# B&R Automation Studio project Morozov_Lab
Automation Studio 

## Logical view

### Library Logical/Libraries/Library (ANSIC)

#### Library.fun - Exported functions and function blocks
```iecst
FUNCTION_BLOCK FB_Controller (*Функциональный блок регулятора*)
	VAR_INPUT
		e : REAL; (*Вход регулятора (об/мин)*)
	END_VAR
	VAR_OUTPUT
		u : REAL; (*Выход регулятора (В)*)
	END_VAR
	VAR
		dt : REAL; (*Шаг интегрирвоания (с)*)
		k_i : REAL; (*Интегральный коэфффициент*)
		k_p : REAL; (*Пропорциональный коэффициент*)
		max_abs_value : REAL; (*Максимальное входное напряжение*)
		integrator : FB_Integrator; (*ФБ-интератор в составе регулятора*)
		iyOld : REAL; (*Разница между выходом регулятора*)
	END_VAR
END_FUNCTION_BLOCK

FUNCTION_BLOCK FB_Integrator (*Функциональный блок интегратора*)
	VAR_INPUT
		in : REAL; (*Вход интеграторируещего звена*)
	END_VAR
	VAR_OUTPUT
		out : REAL; (*Выход интеграторируещего звена*)
	END_VAR
	VAR
		dt : REAL; (*Шаг интегрирования*)
		state : REAL; (*Состояние интегратора на*)
	END_VAR
END_FUNCTION_BLOCK

FUNCTION_BLOCK FB_Motor (*Функциональный блок двигателя*)
	VAR_INPUT
		in : REAL; (*Входное напряжение (В)*)
	END_VAR
	VAR_OUTPUT
		out_w : REAL; (*Частота вращения (об/мин)*)
	END_VAR
	VAR
		dt : REAL; (*Шаг интегрирования (с)*)
		k_e : REAL; (*Постоянная ЭДС двигателя*)
		T_m : REAL; (*Электромеханическая постоянная двигателя*)
		integrator : FB_Integrator; (*ФБ-интегратор в составе двигателя*)
	END_VAR
END_FUNCTION_BLOCK
```

#### FB_Motor.c
```c
#include <bur/plctypes.h>
#ifdef __cplusplus
	extern "C"
	{
#endif
	#include "Library.h"
#ifdef __cplusplus
	};
#endif
/* function block for motors model */
void FB_Motor(struct FB_Motor* inst)
{
	REAL a = inst->in / inst->k_e - inst->out_w;
	REAL b = a / inst->T_m;

	inst->integrator.in = b;
	FB_Integrator(&inst->integrator);

	inst->out_w = inst->integrator.out;
}
```

#### FB_Integrator.c
```c
#include <bur/plctypes.h>
#ifdef __cplusplus
	extern "C"
	{
#endif
	#include "Library.h"
#ifdef __cplusplus
	};
#endif
/* function block for motors model */
void FB_Integrator(struct FB_Integrator* inst)
{
	inst->out=inst->dt * inst ->in+inst->state;
	inst->state=inst->out;
}
```

#### FB_Controller.c
```c
#include <bur/plctypes.h>
#ifdef __cplusplus
	extern "C"
	{
#endif
	#include "Library.h"
#ifdef __cplusplus
	};
#endif
/* TODO: Add your comment here */
void FB_Controller(struct FB_Controller* inst)
{
	REAL a = inst->e * inst->k_p;
	REAL b = inst->e * inst->k_i; // * inst->dt;

	a = a > inst->max_abs_value ? inst->max_abs_value : a;
	a = a < -inst->max_abs_value ? -inst->max_abs_value : a;

	inst->integrator.in = b + inst->iyOld;
	FB_Integrator(&inst->integrator);

	REAL sum = a + inst->integrator.out;

	inst->u = sum;
	inst->u = inst->u > inst->max_abs_value ? inst->max_abs_value : inst->u;
	inst->u = inst->u < -inst->max_abs_value ? -inst->max_abs_value : inst->u;

	inst->iyOld = inst->u - sum;
}
```

#### FB_Regulator.c - not listed in the package file held
```c
#include <bur/plctypes.h>
#ifdef __cplusplus
	extern "C"
	{
#endif
	#include "Library.h"
#ifdef __cplusplus
	};
#endif
/* TODO: Add your comment here */
void FB_Regulator(struct FB_Regulator* inst)
{
	REAL a = inst->in * inst->k_p;
	REAL a = inst->in * inst->k_i; // * inst->dt;

	a = a > inst->max_abs_value ? inst->max_abs_value : a;
	a = a < inst->max_abs_value ? -inst->max_abs_value : a;

	inst->integrator.in = b + inst->iyOld;
	FB_Integrator(&inst->integrator);

	REAL sum = a + inst->integrator.out;

	inst->out = sum;
	inst->out = inst->out > inst->max_abs_value ? inst->max_abs_value : inst->out;
	inst->out = inst->out < -inst->max_abs_value ? -inst->max_abs_value : inst->out;

	inst->iyOld = inst->out - sum;
}
```

### Program Logical/Program

#### Variables.var
```iecst
VAR
	fb_controller : FB_Controller; (*Рассогласование между задающим воздействием и реальной скоростью вращения вала ДПТ [об/мин]*)
	fb_motor : FB_Motor; (*Напряжение, подаваемое на вход 1-го ДПТ [В]*)
	fb_motor2 : FB_Motor; (*Напряжение, подаваемое на вход 2-го ДПТ [В]*)
	speed : REAL; (*Установка по скорости*)
	enable : BOOL; (*Интегральный коэффициент регулятора*)
	counter : REAL; (*Счетчик*)
	fb_integrator : FB_Integrator; (*Интегратор???*)
END_VAR
```

#### Main.cpp
```cpp
#include <bur/plctypes.h>

#ifdef _DEFAULT_INCLUDES
	#include <AsDefault.h>
#endif

// amount of memory to be allocated for heap storage must be specified for every ANSI C++ program with the bur_heap_size variable
unsigned long bur_heap_size = 0xFFFF;

void _INIT ProgramInit(void)
{
	fb_motor.dt = 0.01;
	fb_motor.k_e = 0.24;
	fb_motor.T_m = 0.1;
	fb_motor.in = 0;
	fb_motor.integrator.dt=0.01;

	fb_motor2.dt = 0.01;
	fb_motor2.k_e = 0.24;
	fb_motor2.T_m = 0.1;
	fb_motor2.in = 0;
	fb_motor2.integrator.dt=0.01;

	fb_controller.dt = 0.01;
	fb_controller.integrator.dt = 0.01;
	fb_controller.k_i = 7.2;
	fb_controller.k_p = 0.24 * 3;
	fb_controller.max_abs_value = 24.0;

	speed = 0;
	counter = 0;
	enable = 1;
}

void _CYCLIC ProgramCyclic(void)
{
	if (enable)
	{
		if (counter == 50)
		{
			speed = 50;
		}
		else if (counter == 200)
		{
			speed = 0;
			counter = 0;
		}
		counter++;

		fb_controller.e = speed - fb_motor.out_w;
		FB_Controller(&fb_controller);

		fb_motor.in = fb_controller.u;

		fb_motor2.in = speed * fb_motor2.k_e;

		FB_Motor(&fb_motor);
		FB_Motor(&fb_motor2);
	}
}

void _EXIT ProgramExit(void)
{
	// Insert code here

}
```

Listed in the project but not available here: Logical/Libraries/Library/Types.typ, Logical/Libraries/Library/Constants.var
